Universal Robots PolyScope program: Test ur6c.urp

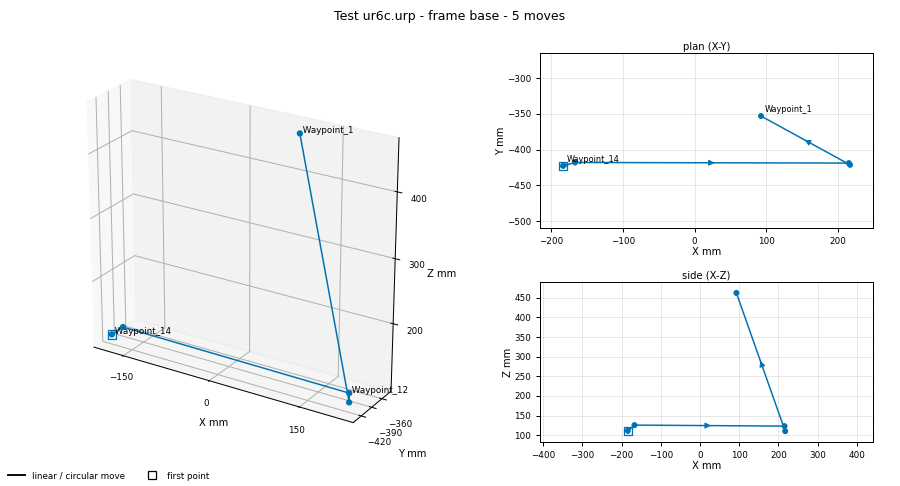
[picture p0: tool path of Test ur6c.urp in frame base, 5 of 5 moves have a stored position in this frame; points joined in program order, loops and branches not executed]
Program Test ur6c (installation=default directory=/programs/usbdisk/NoodleBotSoftware createdIn=3.12.1.90940 lastSavedIn=3.12.1.90940 robotSerialNumber=2017354841)
Calibrated DH parameters: a=[0.000094, -0.006117, -0.382762, 0.000086, 0.000044, 0]; d=[0.089236, 217.751846, -204.357806, -13.283746, 0.094902, 0.082641]; alpha=[1.57017, 0.001953, -0.006493, 1.570192, -1.570543, 0]; deltaTheta=[0.000036, 1.556386, -1.779789, 0.223359, -0.000014, -0.000001]
Robot Program (runOnlyOnce=false)
  MoveL speed 1000 mm/s, acceleration 1200 mm/s^2 (useActiveTCP=true) feature=Base
    Waypoint Waypoint_14: TCP in base x=-183.958 y=-422.781 z=111.127 mm, rx=-2.216 ry=2.1853 rz=0.042 rad; joints [53.402, -90.9, 110.528, 252.259, 268.402, 52.619] deg; flange x=-184.167 y=-430.174 z=297.53 mm, rx=-2.1866 ry=-2.2174 rz=-0.0454 rad
    Wait Sleep waitTime=0.1
    Waypoint Waypoint_13: TCP in base x=-166.927 y=-418.04 z=125.555 mm, rx=2.2093 ry=-2.1712 rz=0.0283 rad; joints [53.613, -96, 114.206, 249.176, 270.389, 52.609] deg; flange x=-163.635 y=-409.814 z=311.952 mm, rx=2.1888 ry=2.2271 rz=-0.0685 rad
    Wait Sleep waitTime=0.1
    Waypoint Waypoint_12: TCP in base x=215.828 y=-418.903 z=123.014 mm, rx=2.1799 ry=-2.2451 rz=0.0047 rad; joints [104.001, -91.491, 109.848, 251.166, 269.185, 105.684] deg; flange x=217.059 y=-416.922 z=309.52 mm, rx=2.2519 ry=2.1864 rz=-0.0191 rad
    Wait Sleep waitTime=0.1
    Waypoint Waypoint_11: TCP in base x=217.45 y=-421.347 z=110.007 mm, rx=-2.1848 ry=2.2499 rz=0.031 rad; joints [103.999, -89.599, 109.567, 251.182, 269.397, 105.681] deg; flange x=219.301 y=-424.69 z=296.552 mm, rx=-2.2396 ry=-2.1747 rz=-0.0082 rad
    URCap RG2 (RG - On Robot, OnRobot A/S) dataModel(depthCompensate=false, force=40, payload=0.0, width=85, name=RG2(85))
    Wait Sleep waitTime=0.1
    Waypoint Waypoint_1: TCP in base x=92.939 y=-353.097 z=462.595 mm, rx=1.1692 ry=-1.2408 rz=1.1709 rad; joints [88.542, -137.018, 138.65, 178.588, 268.341, 89.999] deg; flange x=103.097 y=-166.778 z=463.297 mm, rx=1.2543 ry=1.1818 rz=-1.2438 rad
    Wait Sleep waitTime=0.1
